KUKA KRL program: MeasureConfigStart.src

&ACCESS RVP
&REL 14
DEF MeasureConfigStart ( )

;************************************************
;              CNC Robotics Ltd
;              www.cncrobotics.co.uk
;************************************************
;     Contact: helpdesk@cncrobotics.co.uk
;     Date: 25/09/23
;     Version: 0.13.46
;************************************************
; Description: Program to begin calibration of
; measure sensor
;************************************************

CheckEOATooling(#SPINDLE)
; Enter the tool number, measured lenght and tolerance in the brackets bellow, seperated by commas
ToolMeasureConfig(15,101.40,0.01)

END
